// Brief: Master Arm MasterSlave controller
FUNCTION_BLOCK PUBLIC FB_ArmMasterSlave EXTENDS FB_MasterArmCtrlBase
VAR_INPUT
END_VAR
VAR_OUTPUT
END_VAR
VAR
	// joint4 controller
	m_redunJntCtrl : FB_RedunJntControl;
	
	// flag if project joint4 torque to nullspace
	m_nullspaceCtrl : BOOL :=FALSE;
	

END_VAR

// override this function in each exact controller
METHOD PROTECTED calcCmdJntPos : BOOL
VAR_INPUT
	monitorAngle :LREAL;
	slaveIdx :INT;
END_VAR

VAR_IN_OUT CONSTANT
	i_masterArm :FB_MasterArm;
	i_slaveStatus :ST_SlaveStatus;
END_VAR
var 

END_VAR
m_cmdJntPos:=i_masterArm.curJntPos;
m_cmdJntVel:=i_masterArm.curJntVel;
m_cmdCartPose:=i_masterArm.curCartPose;
END_METHOD

// override this function in each exact controller
METHOD PROTECTED calcCmdJntTrq : BOOL
VAR_input
	monitorAngle :LREAL;
	slaveIdx :INT;
END_VAR

VAR_IN_OUT CONSTANT
	i_masterArm :FB_MasterArm;
	i_slaveStatus :ST_SlaveStatus;
END_VAR

VAR 
	nullspaceMat :Mat7d;
	ctrlTrq : Vec7d;
END_VAR
// redundant joint4 controller
ctrlTrq := g_zeroVec7d;
ctrlTrq[4] := m_redunJntCtrl.run(i_masterArm);

// project to nullspace
IF m_nullspaceCtrl THEN
	nullspaceMat:=i_masterArm.dynaNullspace;
	matMultiVec(nullspaceMat,ctrlTrq, m_cmdJntTrq);
	vecSelfMultiNum(m_cmdJntTrq, ctrlTrq[4] / m_cmdJntTrq[4]);
//	m_cmdJntTrq[5]:=0;
//	m_cmdJntTrq[6]:=0;
//	m_cmdJntTrq[7]:=0;
ELSE
	m_cmdJntTrq := ctrlTrq;
END_IF
END_METHOD

// override this function in each exact controller
// NOTICE: set joint control mode here, and do some initialization if needed
METHOD PUBLIC init : BOOL
VAR_IN_OUT CONSTANT
	i_masterArm	:FB_MasterArm;
END_VAR
VAR_IN_OUT 
	r_masterArmCtrlCmd :ST_ArmCtrlCmds;
END_VAR

VAR
	i:INT;
END_VAR
SUPER^.Init(i_masterArm,r_masterArmCtrlCmd);

m_jntOPMode := g_allTrqMode;

// init controller
m_redunJntCtrl.init(i_masterArm);
END_METHOD

END_FUNCTION_BLOCK

(* stored: Version 1.1.0.1, ProductVersion 3.1.4024.12
   POU FB_ArmMasterSlave: Id {5b96f309-da76-444d-a9fb-2d4321895cd7}, SpecialFunc None
   Method calcCmdJntPos: Id {b549ed00-ec1a-412a-94d0-63a741bf9608}
   Method calcCmdJntTrq: Id {590b7c96-65ed-47d5-8eb2-8a13ee8a5533}
   Method init: Id {1bea1de4-0538-46fc-be44-e671d6da03c3} *)
